Fanuc KAREL source: kt00549.KL

-- PROVISIONAL review KL for V770-1; original PC SHA256 9a26b0e9f32d9514770c58852985ea82c578d7f0351d673df8bd2dd5a2bb2e80
-- Incomplete behavior may be omitted. Consult companion uncertainty JSON. Do not deploy.
PROGRAM KT00549
%NOLOCKGROUP
-- UNRESOLVED_DECL P1 type=000199
-- UNRESOLVED_DECL P2 type=000199
-- UNRESOLVED_DECL OUT type=000101
BEGIN
  -- UNRESOLVED_PC offsets 5-39; opcodes 49,7E,49,7E,60,4A
  -- UNRESOLVED_PC offsets 44-48; opcodes 7F
END KT00549
